(* CODESYS project Text List Example.export

Project tree, tasks and I/O mapping:
  function GetText [ST]
  program Main [ST]
  function block Motor [ST]: ErrorDescription, IsErrorActive
  text list MotorErrorDescriptions
*)

// GetText
FUNCTION GetText : STRING
VAR_INPUT
	textList : STRING;
	id : STRING;
	default : STRING := 'String not found';
END_VAR
VAR
	_result : STRING;
END_VAR


_result := DynamicTextGetDefaultText(ADR(TextList), ADR(Id))^;

GetText := SEL(_result = '', _result, default);

END_FUNCTION

// Main
PROGRAM Main
VAR
	MotorA : Motor;
	ErrorMessage : STRING;	
END_VAR


DynamicTextChangeLanguage('en');

MotorA();

ErrorMessage := MotorA.ErrorDescription;

END_PROGRAM

// Motor
FUNCTION_BLOCK PUBLIC Motor
VAR CONSTANT
	MAX_AMPS : REAL := 100;
	ERROR_DESCRIPTIONS : STRING := 'MotorErrorDescriptions';
END_VAR
VAR
	_motorCurrent : REAL;
	_isActiveError : BOOL;
	_errorDescription : STRING;
END_VAR


IF _motorCurrent > MAX_AMPS THEN
	
	_isActiveError := TRUE;
	
	_errorDescription := GetText(ERROR_DESCRIPTIONS, 'OverCurrent');
	
END_IF

PROPERTY PUBLIC ErrorDescription : STRING
GET

ErrorDescription := _errorDescription;
END_GET
END_PROPERTY

PROPERTY PUBLIC IsErrorActive : BOOL
GET
IsErrorActive := _isActiveError;
END_GET
END_PROPERTY

END_FUNCTION_BLOCK

(* text list MotorErrorDescriptions (id | default)
  OverTemperature | The motor temperature has exceeded safe operating limits.
  OverCurrent | The motor is drawing more current than its rated limit.
  UnderVoltage | The supply voltage is below the acceptable threshold.
   |  *)
